{attribute addProperty BoxType ""}
{attribute addProperty Id "_defaultSyncUnitTasks_486549DC19524.3750DrivesSyncUnitTasks_486549DC19524.3750"}
{attribute addProperty CRC "3587108939"}
{attribute addProperty SizeInBites "390"}
{attribute addProperty SizeInBytes "48.75"}
TYPE SyncUnits_D5CEF04B :
STRUCT
	{attribute addProperty Name "_default"}
	_default : SyncUnitTasks_486549DC;
	{attribute addProperty Name "Drives"}
	Drives : SyncUnitTasks_486549DC;
END_STRUCT
END_TYPE

(* stored: Version 1.2.0.0, ProductVersion 3.1.4024.9
   DUT SyncUnits_D5CEF04B: Id {076380ab-b861-4f9d-ba6a-8436c75fd801} *)
